ABB RobotStudio station: Trainingai4.rsstnx

Station Trainingai4 (saved by RobotStudio 22.2.10013.1)
Controller Trainings5
  mechanical unit ROB_1: IRB4600_60_205_C_01, 6 joints, base frame (0, 0, 0) mm
Layout (positions relative to the parent item):
  - scGripper1 [smart component]
      signals: DI diToolOpen, DI diToolClose, DO doToolOpened, DO doToolClosed, DO doPartPresent
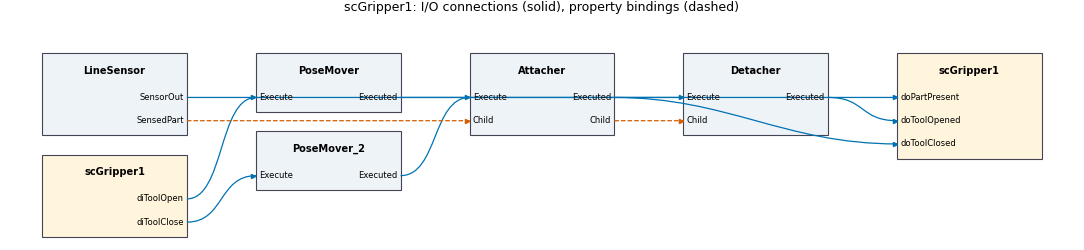
      connections:
        LineSensor.SensorOut -> scGripper1.doPartPresent
        Detacher.Executed -> scGripper1.doToolOpened
        Attacher.Executed -> scGripper1.doToolClosed
        PoseMover.Executed -> Detacher.Execute
        PoseMover_2.Executed -> Attacher.Execute
        scGripper1.diToolOpen -> PoseMover.Execute
        scGripper1.diToolClose -> PoseMover_2.Execute
        LineSensor.SensedPart => Attacher.Child
        Attacher.Child => Detacher.Child
    - LineSensor [smart component, from Components\LineSensor.rslib] at (-7.15, -52.96, 0) mm
        properties: Start=[2.42780829058322 0.0931553945848375 0.59655]; End=[2.376167 0.062155 0.59655]; Radius=0.002; SensedPart=(none); SensedPoint=[0 0 0]
      - _sensorPart_ [part], size 53.7 x 34.4 x 4 mm
    - Attacher [smart component, from Components\Attacher.rslib]
        properties: Parent=(none); Flange=0; Child=(none); Mount=false; Offset=[0 0 0]; Orientation=[0 0 0]
    - Detacher [smart component, from Components\Detacher.rslib]
        properties: Child=(none); KeepPosition=true
    - PoseMover [smart component, from Components\PoseMover.rslib]
        properties: Mechanism=(none); Pose=0; Duration=1
    - PoseMover_2 [smart component, from Components\PoseMover.rslib]
        properties: Mechanism=(none); Pose=2; Duration=1
  - scGripper2 [smart component] at (-1960.6, -1054.27, 0.12) mm
      properties: DetacherChild=(none)
      signals: DI diGripperOpen, DO doGripperOpened, DI diMagnetOn
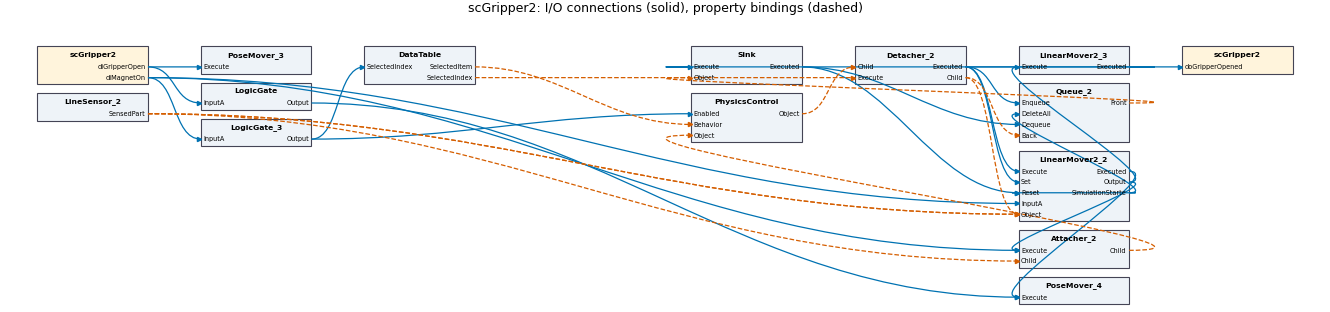
      connections:
        scGripper2.diGripperOpen -> PoseMover_3.Execute
        LinearMover2_2.Executed -> PoseMover_4.Execute
        Detacher_2.Executed -> LinearMover_2.Execute
        LinearMover2_3.Executed -> Sink.Execute
        Detacher_2.Executed -> LogicSRLatch.Set
        LogicSRLatch.Output -> LinearMover2_3.Execute
        Sink.Executed -> LogicSRLatch.Reset
        SimulationEvents_2.SimulationStarted -> LogicSRLatch.Reset
        Detacher_2.Executed -> Queue_2.Enqueue
        SimulationEvents_2.SimulationStarted -> Queue_2.DeleteAll
        Sink.Executed -> Queue_2.Dequeue
        scGripper2.diGripperOpen -> LogicGate.InputA
        LogicGate.Output -> PoseMover_4.Execute
        scGripper2.diMagnetOn -> LogicGate_2.InputA
        LogicGate_2.Output -> Attacher_2.Execute
        scGripper2.diMagnetOn -> Attacher_2.Execute
        scGripper2.diMagnetOn -> LogicGate_3.InputA
        Detacher_2.Executed -> scGripper2.doGripperOpened
        LogicGate_3.Output -> PhysicsControl.Enabled
        LogicGate_3.Output -> DataTable.SelectedIndex
        LineSensor_2.SensedPart => Attacher_2.Child
        LineSensor_2.SensedPart => LinearMover2_2.Object
        LineSensor_2.SensedPart => Positioner_3.Object
        Detacher_2.Child => LinearMover_2.Object
        Detacher_2.Child => Queue_2.Back
        Queue_2.Front => Sink.Object
        DataTable.SelectedItem => PhysicsControl.Behavior
        PhysicsControl.Object => Detacher_2.Child
        Attacher_2.Child => PhysicsControl.Object
        DataTable.SelectedIndex => Detacher_2.Execute
    - LineSensor_2 [smart component, from Components\LineSensor.rslib]
        properties: Start=[1.917656 0.079550000000004 0.234999999999997]; End=[1.917656 0.079550000000004 0.211400999999997]; Radius=0.002; SensedPart=(none); SensedPoint=[0 0 0]
      - _sensorPart_ [part], size 4 x 4 x 23.6 mm
    - PoseMover_3 [smart component, from Components\PoseMover.rslib]
        properties: Mechanism=tGripper2; Pose=2; Duration=0.5
    - PoseMover_4 [smart component, from Components\PoseMover.rslib]
        properties: Mechanism=tGripper2; Pose=0; Duration=0.5
    - Attacher_2 [smart component, from Components\Attacher.rslib]
        properties: Parent=IRB4600_60_205_C_01; Flange=0; Child=(none); Mount=false; Offset=[0 0 0]; Orientation=[0 0 0]
    - Detacher_2 [smart component, from Components\Detacher.rslib]
        properties: Child=(none); KeepPosition=true
    - LogicGate [smart component, from Components\LogicGate.rslib]
        properties: Operator=NOT; Delay=0
    - LogicGate_3 [smart component, from Components\LogicGate.rslib]
        properties: Operator=NOT; Delay=0
    - PhysicsControl [smart component, from Components\PhysicsControl.rslib]
        properties: Object=(none); Behavior=3; SurfaceVelocity=0
    - DataTable [smart component, from Components\DataTable.rslib]
        properties: DataType=Numeric; NumItems=2; SelectedIndex=1; SelectedItem=3; Item0=0; Item1=3
  - IRB4600_60_205_C_01 [mechanism] at (0, 0, 0) mm; joint values [-0.4678, -0.064, 0.6286, 0, 1.0062, -0.4678] (rad or m)
      links: Base, Link1, Link2, Link3, Link4, Link5, Link6
  - extHolder [mechanism] at (-1960.6, -1054.25, 0) mm; joint values [0] (rad or m)
      links: L1, Link
  - tGripper2 [mechanism] at (-42.94, -974.22, 491.53) mm, rotated rx -180 ry 0 rz -90 deg; joint values [1.5708, 1.5708, 1.5708, 1.5708] (rad or m)
      TCP tGripper2 at (0, 187, 0) mm, rotated rx 0 ry -90 rz -90 deg
      links: Baze, Kaire1, Kaire2, Desine1, Desine
  - tGripper1 [mechanism] at (204.61, -1164.7, 660) mm, rotated rx 180 ry 0 rz -150 deg; joint values [0, 0] (rad or m)
      TCP tGripper1 at (0, 85.55, -289) mm, rotated rx 180 ry 0 rz 90 deg
      links: Base, Kaire, Desine
  - scPalletConveyor [smart component]
      connections:
        Source.Executed -> LinearMover2.Execute
        Source.Executed -> Queue.Enqueue
        SimulationEvents.SimulationStarted -> Queue.DeleteAll
        SimulationEvents.SimulationStarted -> Source.Execute
        Source.Copy => LinearMover2.Object
        Source.Copy => Queue.Back
    - LinearMover2 [smart component, from Components\LinearMover2.rslib] at (-2600, 0, 0) mm
        properties: Object=scPalletWithParts_69; Direction=[-0.1 0 0]; Distance=2.6; Duration=5; Reference=Global; ReferenceObject=(none)
    - Source [smart component, from Components\Source.rslib] at (-2600, 0, 0) mm
        properties: Source=scPalletWithParts; Copy=scPalletWithParts_69; Parent=(none); Position=[0 0 0]; Orientation=[0 0 0]; Transient=false; PhysicsBehavior=0
    - scPalletWithParts [smart component] at (-4135.48, 0, -268.92) mm
        connections:
          ParametricBox.GeneratedPart => MatrixRepeater.Source
      - ParametricBox [smart component, from Components\ParametricBox.rslib] at (2772.59, 525, 316.05) mm
          properties: SizeX=0.5; SizeY=0.035; SizeZ=0.015; GeneratedPart=GeneratedPart; KeepGeometry=true
        - GeneratedPart [part], size 500 x 35 x 15 mm
      - MatrixRepeater [smart component, from Components\MatrixRepeater.rslib] at (2768.94, 525, 444) mm
          properties: Source=GeneratedPart; CountX=2; CountY=5; CountZ=1; OffsetX=0.6; OffsetY=0.2; OffsetZ=0.1
        - GeneratedPart [part], size 500 x 35 x 15 mm
        - GeneratedPart [part] at (600, 0, 0) mm, size 500 x 35 x 15 mm
        - GeneratedPart [part] at (0, 200, 0) mm, size 500 x 35 x 15 mm
        - GeneratedPart [part] at (600, 200, 0) mm, size 500 x 35 x 15 mm
        - GeneratedPart [part] at (0, 400, 0) mm, size 500 x 35 x 15 mm
        - GeneratedPart [part] at (600, 400, 0) mm, size 500 x 35 x 15 mm
        - GeneratedPart [part] at (0, 600, 0) mm, size 500 x 35 x 15 mm
        - GeneratedPart [part] at (600, 600, 0) mm, size 500 x 35 x 15 mm
        - GeneratedPart [part] at (0, 800, 0) mm, size 500 x 35 x 15 mm
        - GeneratedPart [part] at (600, 800, 0) mm, size 500 x 35 x 15 mm
      - Solid Face pallet [part] at (2668.87, 425, 300) mm, size 1300 x 1000 x 144 mm
    - Chain Conveyor [part] at (0, 525, 0) mm, size 4159.4 x 900 x 300 mm
    - SimulationEvents [smart component, from Components\SimulationEvents.rslib]
    - Queue [smart component, from Components\Queue.rslib]
        properties: Back=scPalletWithParts_69; Front=scPalletWithParts_69; Queue={e3edb34a-34a1-4ffe-b22b-dbd838811717}; NumberOfObjects=1
    - scPalletWithParts_1 [smart component] at (-2483.52, 0, 0) mm
        connections:
          ParametricBox.GeneratedPart => MatrixRepeater.Source
      - ParametricBox [smart component, from Components\ParametricBox.rslib] at (2772.59, 525, 316.05) mm
          properties: SizeX=0.5; SizeY=0.035; SizeZ=0.015; GeneratedPart=GeneratedPart; KeepGeometry=true
        - GeneratedPart [part], size 500 x 35 x 15 mm
      - MatrixRepeater [smart component, from Components\MatrixRepeater.rslib] at (2768.94, 525, 444) mm
          properties: Source=GeneratedPart; CountX=2; CountY=5; CountZ=1; OffsetX=0.6; OffsetY=0.2; OffsetZ=0.1
        - GeneratedPart [part], size 500 x 35 x 15 mm
        - GeneratedPart [part] at (600, 0, 0) mm, size 500 x 35 x 15 mm
        - GeneratedPart [part] at (0, 200, 0) mm, size 500 x 35 x 15 mm
        - GeneratedPart [part] at (600, 200, 0) mm, size 500 x 35 x 15 mm
        - GeneratedPart [part] at (0, 400, 0) mm, size 500 x 35 x 15 mm
        - GeneratedPart [part] at (600, 400, 0) mm, size 500 x 35 x 15 mm
        - GeneratedPart [part] at (0, 600, 0) mm, size 500 x 35 x 15 mm
        - GeneratedPart [part] at (600, 600, 0) mm, size 500 x 35 x 15 mm
        - GeneratedPart [part] at (0, 800, 0) mm, size 500 x 35 x 15 mm
        - GeneratedPart [part] at (600, 800, 0) mm, size 500 x 35 x 15 mm
    - scPalletWithParts_24 [smart component] at (-2600, 0, 0) mm
        connections:
          ParametricBox.GeneratedPart => MatrixRepeater.Source
      - ParametricBox [smart component, from Components\ParametricBox.rslib] at (2772.59, 525, 316.05) mm
          properties: SizeX=0.5; SizeY=0.035; SizeZ=0.015; GeneratedPart=GeneratedPart; KeepGeometry=true
        - GeneratedPart [part], size 500 x 35 x 15 mm
      - MatrixRepeater [smart component, from Components\MatrixRepeater.rslib] at (2768.94, 525, 444) mm
          properties: Source=GeneratedPart; CountX=2; CountY=5; CountZ=1; OffsetX=0.6; OffsetY=0.2; OffsetZ=0.1
        - GeneratedPart [part], size 500 x 35 x 15 mm
        - GeneratedPart [part] at (600, 0, 0) mm, size 500 x 35 x 15 mm
        - GeneratedPart [part] at (0, 200, 0) mm, size 500 x 35 x 15 mm
        - GeneratedPart [part] at (600, 200, 0) mm, size 500 x 35 x 15 mm
        - GeneratedPart [part] at (0, 400, 0) mm, size 500 x 35 x 15 mm
        - GeneratedPart [part] at (600, 400, 0) mm, size 500 x 35 x 15 mm
        - GeneratedPart [part] at (0, 600, 0) mm, size 500 x 35 x 15 mm
        - GeneratedPart [part] at (600, 600, 0) mm, size 500 x 35 x 15 mm
        - GeneratedPart [part] at (0, 800, 0) mm, size 500 x 35 x 15 mm
        - GeneratedPart [part] at (600, 800, 0) mm, size 500 x 35 x 15 mm
    - scPalletWithParts_41 [smart component] at (-2600, 0, 0) mm
        connections:
          ParametricBox.GeneratedPart => MatrixRepeater.Source
      - ParametricBox [smart component, from Components\ParametricBox.rslib] at (2772.59, 525, 316.05) mm
          properties: SizeX=0.5; SizeY=0.035; SizeZ=0.015; GeneratedPart=GeneratedPart; KeepGeometry=true
        - GeneratedPart [part], size 500 x 35 x 15 mm
      - MatrixRepeater [smart component, from Components\MatrixRepeater.rslib] at (2768.94, 525, 444) mm
          properties: Source=GeneratedPart; CountX=2; CountY=5; CountZ=1; OffsetX=0.6; OffsetY=0.2; OffsetZ=0.1
        - GeneratedPart [part], size 500 x 35 x 15 mm
        - GeneratedPart [part] at (600, 0, 0) mm, size 500 x 35 x 15 mm
        - GeneratedPart [part] at (0, 200, 0) mm, size 500 x 35 x 15 mm
        - GeneratedPart [part] at (600, 200, 0) mm, size 500 x 35 x 15 mm
        - GeneratedPart [part] at (0, 400, 0) mm, size 500 x 35 x 15 mm
        - GeneratedPart [part] at (600, 400, 0) mm, size 500 x 35 x 15 mm
        - GeneratedPart [part] at (0, 600, 0) mm, size 500 x 35 x 15 mm
        - GeneratedPart [part] at (600, 600, 0) mm, size 500 x 35 x 15 mm
        - GeneratedPart [part] at (0, 800, 0) mm, size 500 x 35 x 15 mm
        - GeneratedPart [part] at (600, 800, 0) mm, size 500 x 35 x 15 mm
      - Solid Face pallet [part] at (2668.87, 425, 300) mm, size 1300 x 1000 x 144 mm
    - scPalletWithParts_69 [smart component] at (-2600, 0, 0) mm
        connections:
          ParametricBox.GeneratedPart => MatrixRepeater.Source
      - ParametricBox [smart component, from Components\ParametricBox.rslib] at (2772.59, 525, 316.05) mm
          properties: SizeX=0.5; SizeY=0.035; SizeZ=0.015; GeneratedPart=GeneratedPart; KeepGeometry=true
        - GeneratedPart [part], size 500 x 35 x 15 mm
      - MatrixRepeater [smart component, from Components\MatrixRepeater.rslib] at (2768.94, 525, 444) mm
          properties: Source=GeneratedPart; CountX=2; CountY=5; CountZ=1; OffsetX=0.6; OffsetY=0.2; OffsetZ=0.1
        - GeneratedPart [part], size 500 x 35 x 15 mm
        - GeneratedPart [part] at (600, 0, 0) mm, size 500 x 35 x 15 mm
        - GeneratedPart [part] at (0, 200, 0) mm, size 500 x 35 x 15 mm
        - GeneratedPart [part] at (600, 200, 0) mm, size 500 x 35 x 15 mm
        - GeneratedPart [part] at (0, 400, 0) mm, size 500 x 35 x 15 mm
        - GeneratedPart [part] at (600, 400, 0) mm, size 500 x 35 x 15 mm
        - GeneratedPart [part] at (0, 600, 0) mm, size 500 x 35 x 15 mm
        - GeneratedPart [part] at (600, 600, 0) mm, size 500 x 35 x 15 mm
        - GeneratedPart [part] at (0, 800, 0) mm, size 500 x 35 x 15 mm
        - GeneratedPart [part] at (600, 800, 0) mm, size 500 x 35 x 15 mm
      - Solid Face pallet [part] at (2668.87, 425, 300) mm, size 1300 x 1000 x 144 mm
  - scPartConveyor [smart component]
      properties: DetacherChild=(none)
      signals: DI diGripperOpened
      connections:
        SimulationEvents_2.SimulationStarted -> Queue_2.DeleteAll
        LinearMover2_3.Executed -> Sink.Execute
        Sink.Executed -> Queue_2.Dequeue
        scPartConveyor.diGripperOpened -> Queue_2.Enqueue
        Timer.Output -> LinearMover2_3.Execute
        scPartConveyor.diGripperOpened -> Timer.Active
        scPartConveyor.diGripperOpened -> LinearMover2_3.Execute
        scPartConveyor.DetacherChild => Queue_2.Back
    - Belt Conveyor [part] at (1257.28, -128.32, 0) mm, rotated rx 0 ry 0 rz -90 deg, size 5091 x 400 x 600 mm
    - Sink [smart component, from Components\Sink.rslib]
        properties: Object=(none)
    - Queue_2 [smart component, from Components\Queue.rslib]
        properties: Back=(none); Front=(none); Queue={c67b11fc-2095-4afd-a85c-1ddee9b4cd59};{708fda7a-92f7-4d05-9491-8615157d7df2};{67461ff7-22f6-4c29-9fed-22203bfd249f};{64e9e6e7-333e-4201-933d-d7f85a6942f3};{94ed0397-e4d9-4dbd-8b65-1c47b80f1687};{0e5ceeee-6866-4557-879f-678caf6cbf5d};{c77d8a7a-4c8b-4a63-93cd-95f10a3ba390};{2dc8e61b-ebec-44af-ad14-0ed559f0599e};{a771ce6e-0ae6-4e53-ab8f-f897429e7bdc};{55db3552-5567-4b7d-9fc8-0461d874dd02};{eca2981a-a2f0-4461-8ce5-34812ac5fa19};{0c85abd3-7812-48b3-ae52-80a0c9b890cb};{4e699870-b5d5-45c6-8165-44d45a72ec64};{717bbeb6-b8bc-4b00-a186-3d805d64528c};{651f6ac5-aea8-47f9-ae17-ed7998c333a4};{7c32ac3b-945e-400d-8ce3-24234b8ee495};{71834a44-749a-4cb6-8886-d85a4c408215};{7ab371d3-c5f9-41aa-aa14-6d825ef1be4f};{28583303-bd4f-4e9c-906b-fdd82cf9f385};{6c8c032e-3ace-4d8c-9ade-9f0e9220f704};{53d18044-a4a6-47e9-a2fd-a88179a397c4};{f98f4791-6472-4895-9234-1f3cf1dbf26f};{76240e30-d61d-432f-bdfa-ab9751f1b838};{3e2c236a-aa4f-4aca-a898-b86b4838ce87};{8efbb0bd-58a3-4156-8114-2d818540220e};{383bef30-bc5f-4f9a-83c2-b0e34f40491d};{85feea3d-e578-435b-8a0a-43b224609656};{7d6159f7-02fe-4613-abe4-c9ae4e2f11ab};{33503d57-5cf7-4ece-aeb4-f011f00fb54d};{af74fe30-0894-4f1b-9fbe-9a7e2716110b};{af57b412-42c3-4c7b-8199-7909dbcf08f4};{018e3041-176c-43ec-8c03-727afeb9b32d};{8be667fe-11ba-4109-9375-b98e5219bea1};{d23d0b7f-f891-4a8f-bfba-fc5707fab13a};{b891840e-4aac-46b0-8260-738cb80d5b75};{fa70ff57-8a2c-476f-9041-d0400eecf8eb};{9c520f9e-5298-43dc-b2a8-0cb615bae637};{60e750eb-7b52-474d-ae52-ff52f4173b29};{2e5c8f01-c4b5-456c-9932-b4f5dee0107b};{7cc00504-0dce-4288-9317-d0d6fe0c5c7c};{a5f28ec1-5dc2-4ed1-8193-ab70b21bbfdf};{ce9ec1a0-0e60-4302-a700-a5878b59edd3};{793488a4-99cf-42ff-aac9-6560d6ab3dd0};{78454220-a91c-468d-8c3c-db103b123668};{05bacae4-9263-4ba8-b032-70854a68714a};{bcc7de2b-fc59-4f15-89ab-b5e14cbe93ed};{9891b9ae-2fa4-4f68-964b-9ce407872076};{d7a565d5-c072-4b25-882f-d1a2a52e6e9c};{434aaa15-53f6-4512-a66b-7f3fe4fc45fe};{71fa1183-a7c1-4c06-a958-2085be59233c};{ee92a2f4-ddd4-4dd9-a94a-1fa7b2ea8aa9};{1017cba6-3294-4f27-a96c-eb482c7965fe};{6d9c7b12-6d72-467e-b8a3-be2238fcecf5};{4b882337-32f4-4e0a-87d2-8f2db3b9d2e8};{253ddf78-036f-4a0f-90da-56371ce81ddd};{49d3ad0f-bb53-484d-95c5-53db075cda27};{82c4a3c8-fc2f-4837-ae14-c5e6bbde5f68};{7d816fb5-cfba-4278-889c-cd7513db15b4};{b3b80dac-fe28-4e9a-a3b7-89359c8b250d};{ce33794c-e366-4e3b-968e-b1c013470eb6};{9a010937-6ca3-4c8e-b239-b6e2c5ada9a5};{ac9e126c-4771-45ed-b637-2080433cdff7};{87beb8d5-ea09-4810-bced-b4155644339e};{5d5839d6-3185-4b06-9573-46cd0e03e8d5};{9efd49b7-ab8d-4944-b626-336959d1e523};{bc1d41b0-9db8-423c-9e97-e9e43a1e4657};{22a1b044-18e0-472a-a9e1-30924429c904};{d83b3222-dc2f-41dc-b778-deba45f1b867};{377c1028-79fd-4e9a-99e1-5e1dabc565dc};{ccad18d2-834a-473c-9ada-c504c03ebbb5};{d93c8256-e4a3-4ca3-bbc5-00eccdd6f70c};{c4cb70a9-ed40-4b39-be76-fa0083d9cb71};{2a2b9da9-6ac0-4114-9e8a-7ffa9b42bd76};{a03b483c-f943-4b98-a38b-b284bb909042};{480dbded-ecbf-4194-b014-7a86e9249e95};{1624253f-d864-4b0e-9380-399f05db383b};{728b13e3-94af-45f1-8693-04a85384dff7};{1ee0b563-f1ac-456a-ac4f-51b5b1871d4d};{2f9643c4-2f89-4d7f-9f3e-4f8bd829e7cd};{e4538fc9-f0e2-4ad0-81b0-c7d0ce9b22f3};{d58af41f-3b5e-4606-a58b-32e085b97b09};{a1b85fca-56a0-4999-940a-3313be6c515a};{9b39818f-9239-4860-80d9-1377808265c3};{71c3e6b7-6229-42e7-ae5d-48cc175b6e3a};{8f26967d-2560-4642-ba05-c3230d003f64};{12a119c8-c476-4974-aa3f-296f0bdf2b6d};{e969b842-8b65-45d0-8057-a9c2f9d6e45c};{a891d8ce-4a65-44a3-b847-c242bb7fd2b4};{e5dcd1f9-d137-4374-95a7-e6480d10f156};{7e4cee50-cf00-4268-8c89-27e3d911d00a};{55853810-ede1-4308-bec4-0666d8f9d3f3};{0136c5c5-1471-4a9b-96db-006ea4bb1f89};{5243cab9-d156-446e-b45a-fc89aa48f761};{d4ae2440-03e7-4030-9d9d-accdd5b969e0};{7666d739-cf43-42a6-bfcd-22210b3e0e0b};{57bed969-b163-4791-92ff-c22e541c3b98};{f51b92c4-83eb-4967-b9d8-464ebb6ed4f1};{640ae70b-27e3-4432-bc9c-546c6403e958};{a4a47a1e-a2fd-4bc4-a667-b5c91d247590};{f263b00d-b872-44a0-877c-010eb61af663};{efa0d8d9-c0b0-401e-bfcb-857f42b7fa40};{eafabbec-0366-4c69-8d76-a39271a541f2};{201a7442-acd4-4ea5-bada-7e46e4445394};{ebd8d3ad-9e11-4c86-b649-7f76f6f19318};{0f75645c-cd97-460b-a6df-c8ed1b7c9322}; NumberOfObjects=0
    - LinearMover2_3 [smart component, from Components\LinearMover2.rslib]
        properties: Object=Queue_2; Direction=[0 -4.5 0]; Distance=4; Duration=5; Reference=Global; ReferenceObject=(none)
  - scToolChanger [smart component]
      signals: DI diAttachTool, DI diDetachTool
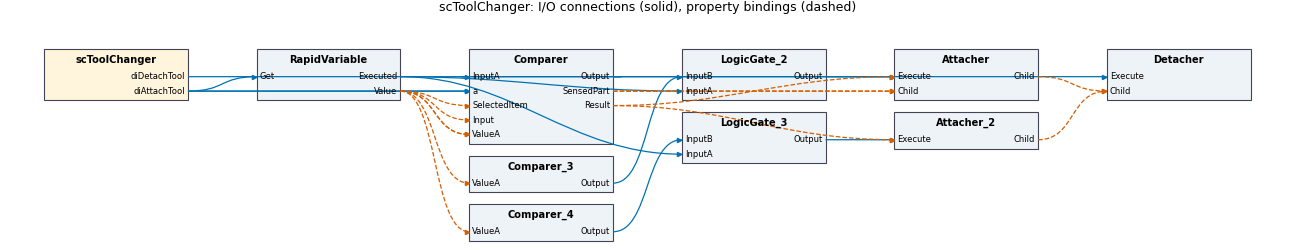
      connections:
        scToolChanger.diDetachTool -> Detacher.Execute
        scToolChanger.diAttachTool -> RapidVariable.Get
        Comparer.Output -> Attacher.Execute
        Comparer.Output -> LogicGate.InputA
        scToolChanger.diAttachTool -> Expression_2.a
        scToolChanger.diAttachTool -> Expression.a
        Comparer_3.Output -> LogicGate_2.InputB
        LogicGate_2.Output -> Attacher.Execute
        Comparer_4.Output -> LogicGate_3.InputB
        LogicGate_3.Output -> Attacher_2.Execute
        RapidVariable.Executed -> LogicGate_3.InputA
        RapidVariable.Executed -> LogicGate_2.InputA
        LineSensor.SensedPart => Attacher.Child
        Attacher.Child => Detacher.Child
        VolumeSensor.SensedPart => Attacher.Child
        RapidVariable.Value => DataTable_3.SelectedItem
        RapidVariable.Value => LogicSplit.Input
        Attacher_2.Child => Detacher.Child
        RapidVariable.Value => Comparer.ValueA
        RapidVariable.Value => Comparer_2.ValueA
        Expression.Result => Attacher.Execute
        Expression_2.Result => Attacher_2.Execute
        RapidVariable.Value => Comparer_3.ValueA
        RapidVariable.Value => Comparer_4.ValueA
    - Swivel [part] at (912.28, -460.91, 892.32) mm, rotated rx 180 ry 0 rz 180 deg, size 181 x 209 x 109.7 mm
    - Attacher [smart component, from Components\Attacher.rslib]
        properties: Parent=IRB4600_60_205_C_01; Flange=0; Child=tGripper2; Mount=true; Offset=[0 0 0]; Orientation=[0 0 0]
    - Detacher [smart component, from Components\Detacher.rslib]
        properties: Child=tGripper1; KeepPosition=false
    - RapidVariable [smart component, from Components\RapidVariable.rslib]
        properties: DataType=num; Controller=Trainings5; Task=T_ROB1; Module=Main_; Variable=nWhichTool; Value=1
    - Attacher_2 [smart component, from Components\Attacher.rslib]
        properties: Parent=IRB4600_60_205_C_01; Flange=0; Child=tGripper1; Mount=true; Offset=[0 0 0]; Orientation=[0 0 0]
    - Comparer_3 [smart component, from Components\Comparer.rslib]
        properties: ValueA=1; Operator===; ValueB=2
    - Comparer_4 [smart component, from Components\Comparer.rslib]
        properties: ValueA=1; Operator===; ValueB=1
    - LogicGate_2 [smart component, from Components\LogicGate.rslib]
        properties: Operator=AND; Delay=0
    - LogicGate_3 [smart component, from Components\LogicGate.rslib]
        properties: Operator=AND; Delay=0
  - Belt Conveyor [part] at (1083.59, -3149.63, 0) mm, rotated rx 0 ry 0 rz 90 deg, size 3091 x 400 x 600 mm
  - Part_2 [part] at (-180.97, -2987.59, 0) mm, size 400 x 3000 x 2 mm
Attachment: Swivel is attached to IRB4600_60_205_C_01 / Link6
Attachment: scGripper2 is attached to tGripper2 / Baze
Attachment: T8147_055 flan_as susiaurintam is attached to IRB4600_60_205_C_01 / Link6
Attachment: scGripper1 is attached to Attacher
Station logic (signal -> signal, property => property):
  scGripper2.doGripperOpened -> scPartConveyor.diGripperOpened
  Trainings5.doGripper2Open -> scGripper2.diGripperOpen
  Trainings5.doMagnetOn -> scGripper2.diMagnetOn
  Trainings5.doAttachTool -> scToolChanger.diAttachTool
  Trainings5.doDetachTool -> scToolChanger.diDetachTool
  scGripper2.DetacherChild => scPartConveyor.DetacherChild
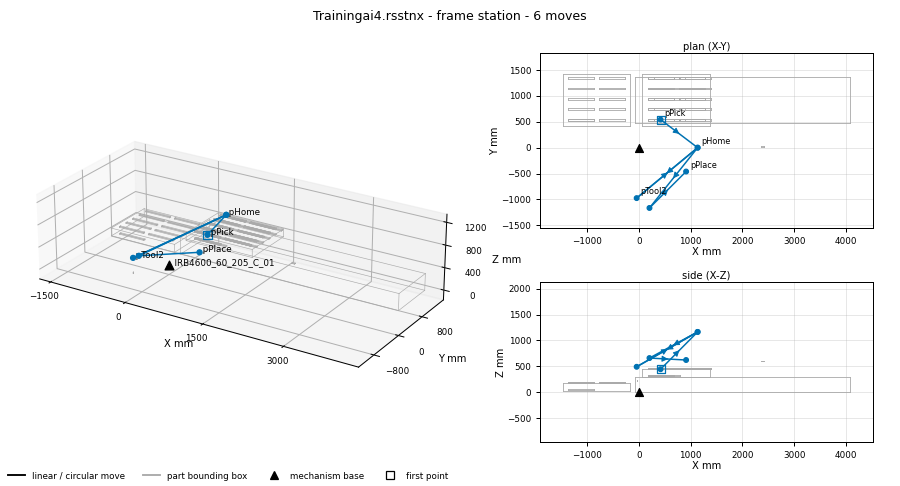
[picture p0: tool path of Trainingai4.rsstnx in frame station, 6 of 6 moves have a stored position in this frame; points joined in program order, loops and branches not executed]
Targets, tools, work objects and paths stored in the station, written as RAPID:
! task T_ROB1
MODULE CalibData
  PERS tooldata tGripper1:=[TRUE,[[-289,0,168.55],[1,0,0,0]],[5,[0,0,100],[1,0,0,0],0,0,0]];
  PERS tooldata tGripper2:=[TRUE,[[0,0,172.001],[1,0,0,0]],[3,[0,0,100],[1,0,0,0],0,0,0]];
ENDMODULE

! task T_ROB1
MODULE CalibData
  TASK PERS wobjdata wPallet:=[FALSE,TRUE,"",[[68.866,424.996,300],[1,0,0,0]],[[0,0,0],[1,0,0,0]]];
  CONST robtarget pPick:=[[350.075,117.5,144],[0,-0.707106781,0.707106781,0],[0,0,-1,0],[9E+09,9E+09,9E+09,9E+09,9E+09,9E+09]];
  PERS tooldata tGripper2:=[TRUE,[[0,0,270],[1,0,0,0]],[3,[0,0,100],[1,0,0,0],0,0,0]];
  CONST robtarget pHome:=[[1135,0,1165],[0,0,1,0],[0,0,0,0],[9E+09,9E+09,9E+09,9E+09,9E+09,9E+09]];
  CONST robtarget pPlace:=[[912.278592303,-460.91,622.316100316],[0,0,1,0],[0,0,0,0],[9E+09,9E+09,9E+09,9E+09,9E+09,9E+09]];
  PERS tooldata tGripper1:=[TRUE,[[-289,0,168.55],[0.707106781,0,-0.707106781,0]],[5,[0,0,100],[1,0,0,0],0,0,0]];
  PROC Path_10()
    MoveL pPick,v1000,z100,tGripper2\WObj:=wPallet;
    MoveL pHome,v1000,z100,tGripper2\WObj:=wobj0;
    MoveL pTool2,v1000,z100,tool0\WObj:=wobj0;
    MoveL pHome,v1000,z100,tGripper2\WObj:=wobj0;
    MoveL pTool1,v1000,z100,tool0\WObj:=wobj0;
    MoveL pPlace,v1000,z100,tGripper2\WObj:=wobj0;
  ENDPROC
ENDMODULE

! task T_ROB1
MODULE Module1
  CONST robtarget pTool2:=[[-42.943005524,-974.204110584,491.401],[0,-0.707106781,0.707106781,0],[-2,0,-3,0],[9E+09,9E+09,9E+09,9E+09,9E+09,9E+09]];
  CONST robtarget pTool1:=[[204.606994476,-1164.704110584,660],[0,-0.258819045,0.965925826,0],[-1,0,-2,0],[9E+09,9E+09,9E+09,9E+09,9E+09,9E+09]];
ENDMODULE

